FUNCTION WRITE_ANY_REAL : BOOL
VAR_INPUT
    ptr: POINTER TO REAL;
    val: REAL;
END_VAR

ptr^ := val;

END_FUNCTION

(* stored: Version 1.1.0.1, ProductVersion 3.1.4022.9
   POU WRITE_ANY_REAL: Id {b51bba4d-2ead-4155-a62f-7a7ea20f8571}, SpecialFunc None *)
